FUNCTION_BLOCK FB_RunClock
VAR_INPUT
	bStart 		: BOOL;
	bStop 		: BOOL;
	fCycleTime  : LREAL;
END_VAR
VAR_OUTPUT
	fTime : LREAL;
END_VAR
VAR
	bOnOff : BOOL;
END_VAR

IF bStop OR (G_Work.eStatus = E_Status.Off) THEN
	bOnOff := FALSE;
	fTime := 0.0;
ELSIF bOnOff OR bStart AND (G_Work.eStatus = E_Status.Starting) THEN
	bOnOff := TRUE;
	fTime := fTime + fCycleTime;
END_IF

END_FUNCTION_BLOCK

(* stored: Version 1.1.0.1, ProductVersion 3.1.4024.12
   POU FB_RunClock: Id {72885421-59e1-4582-bbdc-64c324631609}, SpecialFunc None *)
